	        REGION CATHODE PNP X1 FWD OUTPUT CAM
	            #tempOutputCam ?= #OutputCam.CathodePnPX1FwdOutputCam;
	            #instResetCathodePnPX1FwdOutputCam(Axis := #tempOutputCam^,
	                                               Execute := #statNowCmd = #STAT_RESET,
	                                               Restart:= NOT #tempOutputCam^.StatusWord.%X0);
	        END_REGION

	        REGION CATHODE PNP X1 BWD OUTPUT CAM
	            #tempOutputCam ?= #OutputCam.CathodePnPX1BwdOutputCam;
	            #instResetCathodePnPX1BwdOutputCam(Axis := #tempOutputCam^,
	                                               Execute := #statNowCmd = #STAT_RESET,
	                                               Restart:= NOT #tempOutputCam^.StatusWord.%X0);
	        END_REGION

	        REGION CATHODE PNP X2 FWD OUTPUT CAM
	            #tempOutputCam ?= #OutputCam.CathodePnPX2FwdOutputCam;
	            #instResetCathodePnPX2FwdOutputCam(Axis := #tempOutputCam^,
	                                               Execute := #statNowCmd = #STAT_RESET,
	                                               Restart:= NOT #tempOutputCam^.StatusWord.%X0);
	        END_REGION

	        REGION CATHODE PNP X2 BWD OUTPUT CAM
	            #tempOutputCam ?= #OutputCam.CathodePnPX2BwdOutputCam;
	            #instResetCathodePnPX2BwdOutputCam(Axis := #tempOutputCam^,
	                                               Execute := #statNowCmd = #STAT_RESET,
	                                               Restart:= NOT #tempOutputCam^.StatusWord.%X0);
	        END_REGION

	        REGION CATHODE PNP Z1 DOWN 1 OUTPUT CAM
	            #tempOutputCam ?= #OutputCam.CathodePnPZ1Down1OutputCam;
	            #instResetCathodePnPZ1Down1OutputCam(Axis := #tempOutputCam^,
	                                                 Execute := #statNowCmd = #STAT_RESET,
	                                                 Restart:= NOT #tempOutputCam^.StatusWord.%X0);
	        END_REGION

	        REGION CATHODE PNP Z1 UP 1 OUTPUT CAM
	            #tempOutputCam ?= #OutputCam.CathodePnPZ1Up1OutputCam;
	            #instResetCathodePnPZ1Up1OutputCam(Axis := #tempOutputCam^,
	                                               Execute := #statNowCmd = #STAT_RESET,
	                                               Restart:= NOT #tempOutputCam^.StatusWord.%X0);
	        END_REGION

	        REGION CATHODE PNP Z2 DOWN 1 OUTPUT CAM
	            #tempOutputCam ?= #OutputCam.CathodePnPZ2Down1OutputCam;
	            #instResetCathodePnPZ2Down1OutputCam(Axis := #tempOutputCam^,
	                                                 Execute := #statNowCmd = #STAT_RESET,
	                                                 Restart:= NOT #tempOutputCam^.StatusWord.%X0);
	        END_REGION

	        REGION CATHODE PNP Z2 UP 1 OUTPUT CAM
	            #tempOutputCam ?= #OutputCam.CathodePnPZ2Up1OutputCam;
	            #instResetCathodePnPZ2Up1OutputCam(Axis := #tempOutputCam^,
	                                               Execute := #statNowCmd = #STAT_RESET,
	                                               Restart:= NOT #tempOutputCam^.StatusWord.%X0);
	        END_REGION

	        REGION CATHODE PNP Z1 DOWN 2 OUTPUT CAM
	            #tempOutputCam ?= #OutputCam.CathodePnPZ1Down2OutputCam;
	            #instResetCathodePnPZ1Down2OutputCam(Axis := #tempOutputCam^,
	                                                 Execute := #statNowCmd = #STAT_RESET,
	                                                 Restart:= NOT #tempOutputCam^.StatusWord.%X0);
	        END_REGION

	        REGION CATHODE PNP Z1 UP 2 OUTPUT CAM
	            #tempOutputCam ?= #OutputCam.CathodePnPZ1Up2OutputCam;
	            #instResetCathodePnPZ1Up2OutputCam(Axis := #tempOutputCam^,
	                                               Execute := #statNowCmd = #STAT_RESET,
	                                               Restart:= NOT #tempOutputCam^.StatusWord.%X0);
	        END_REGION

	        REGION CATHODE PNP Z2 DOWN 2 OUTPUT CAM
	            #tempOutputCam ?= #OutputCam.CathodePnPZ2Down2OutputCam;
	            #instResetCathodePnPZ2Down2OutputCam(Axis := #tempOutputCam^,
	                                                 Execute := #statNowCmd = #STAT_RESET,
	                                                 Restart:= NOT #tempOutputCam^.StatusWord.%X0);
	        END_REGION

	        REGION CATHODE PNP Z2 UP 2 OUTPUT CAM
	            #tempOutputCam ?= #OutputCam.CathodePnPZ2Up2OutputCam;
	            #instResetCathodePnPZ2Up2OutputCam(Axis := #tempOutputCam^,
	                                               Execute := #statNowCmd = #STAT_RESET,
	                                               Restart:= NOT #tempOutputCam^.StatusWord.%X0);
	        END_REGION

	        REGION CATHODE PNP Z1 SUCTION ON OUTPUT CAM
	            #tempOutputCam ?= #OutputCam.CathodePnPZ1SuctionOnOutputCam;
	            #instResetCathodePnPZ1SuctionOnOutputCam(Axis := #tempOutputCam^,
	                                                     Execute := #statNowCmd = #STAT_RESET,
	                                                     Restart:= NOT #tempOutputCam^.StatusWord.%X0);
	        END_REGION

	        REGION CATHODE PNP Z1 SUCTION OFF OUTPUT CAM
	            #tempOutputCam ?= #OutputCam.CathodePnPZ1SuctionOffOutputCam;
	            #instResetCathodePnPZ1SuctionOffOutputCam(Axis := #tempOutputCam^,
	                                                      Execute := #statNowCmd = #STAT_RESET,
	                                                      Restart:= NOT #tempOutputCam^.StatusWord.%X0);
	        END_REGION

	        REGION CATHODE PNP Z1 REEL CUT BLOW OUTPUT CAM
	            #tempOutputCam ?= #OutputCam.CathodePnPZ1ReelCutBlowOutputCam;
	            #instResetCathodePnPZ1ReelCutBlowOutputCam(Axis := #tempOutputCam^,
	                                                       Execute := #statNowCmd = #STAT_RESET,
	                                                       Restart:= NOT #tempOutputCam^.StatusWord.%X0);
	        END_REGION

	        REGION CATHODE PNP Z2 SUCTION ON OUTPUT CAM
	            #tempOutputCam ?= #OutputCam.CathodePnPZ2SuctionOnOutputCam;
	            #instResetCathodePnPZ2SuctionOnOutputCam(Axis := #tempOutputCam^,
	                                                     Execute := #statNowCmd = #STAT_RESET,
	                                                     Restart:= NOT #tempOutputCam^.StatusWord.%X0);
	        END_REGION

	        REGION CATHODE PNP Z2 SUCTION OFF OUTPUT CAM
	            #tempOutputCam ?= #OutputCam.CathodePnPZ2SuctionOffOutputCam;
	            #instResetCathodePnPZ2SuctionOffOutputCam(Axis := #tempOutputCam^,
	                                                      Execute := #statNowCmd = #STAT_RESET,
	                                                      Restart:= NOT #tempOutputCam^.StatusWord.%X0);
	        END_REGION

	        REGION CATHODE ALIGN SUCTION ON OUTPUT CAM
	            #tempOutputCam ?= #OutputCam.CathodeAlignSuctionOnOutputCam;
	            #instResetCathodeAlignSuctionOnOutputCam(Axis := #tempOutputCam^,
	                                                     Execute := #statNowCmd = #STAT_RESET,
	                                                     Restart:= NOT #tempOutputCam^.StatusWord.%X0);
	        END_REGION

	        REGION CATHODE ALIGN SUCTION OFF OUTPUT CAM
	            #tempOutputCam ?= #OutputCam.CathodeAlignSuctionOffOutputCam;
	            #instResetCathodeAlignSuctionOffOutputCam(Axis := #tempOutputCam^,
	                                                      Execute := #statNowCmd = #STAT_RESET,
	                                                      Restart:= NOT #tempOutputCam^.StatusWord.%X0);
	        END_REGION

	        REGION FINAL ROLLER X FWD OUTPUT CAM
	            #tempOutputCam ?= #OutputCam.FinalRollerXFwdOutputCam;
	            #instResetFinalRollerXFwdOutputCam(Axis := #tempOutputCam^,
	                                               Execute := #statNowCmd = #STAT_RESET,
	                                               Restart := NOT #tempOutputCam^.StatusWord.%X0);
	        END_REGION

	        REGION FINAL ROLLER X BWD OUTPUT CAM
	            #tempOutputCam ?= #OutputCam.FinalRollerXBwdOutputCam;
	            #instResetFinalRollerXBwdOutputCam(Axis := #tempOutputCam^,
	                                               Execute := #statNowCmd = #STAT_RESET,
	                                               Restart := NOT #tempOutputCam^.StatusWord.%X0);
	        END_REGION

	        REGION FINAL ROLLER X STACK TABLE DOWN OUTPUT CAM
	            #tempOutputCam ?= #OutputCam.FinalRollerXStackTableDownOutputCam;
	            #instResetFinalRollerXStackTableDownOutputCam(Axis := #tempOutputCam^,
	                                                          Execute := #statNowCmd = #STAT_RESET,
	                                                          Restart := NOT #tempOutputCam^.StatusWord.%X0);
	        END_REGION

	        REGION FINAL ROLLER X STACK ANODE VISION OUTPUT CAM
	            #tempOutputCam ?= #OutputCam.FinalRollerXStackAnodeVisionOutputCam;
	            #instResetFinalRollerXStackAnodeVisionOutputCam(Axis := #tempOutputCam^,
	                                                            Execute := #statNowCmd = #STAT_RESET,
	                                                            Restart := NOT #tempOutputCam^.StatusWord.%X0);
	        END_REGION

	        REGION FINAL ROLLER X STACK CATHODE VISION OUTPUT CAM
	            #tempOutputCam ?= #OutputCam.FinalRollerXStackCathodeVisionOutputCam;
	            #instResetFinalRollerXStackCathodeVisionOutputCam(Axis := #tempOutputCam^,
	                                                              Execute := #statNowCmd = #STAT_RESET,
	                                                              Restart := NOT #tempOutputCam^.StatusWord.%X0);
	        END_REGION

	        REGION ANODE PNP Z1 REEL CUT DATA DELETE ON OUTPUT CAM
	            #tempOutputCam ?= #OutputCam.AnodePnPZ1ReelCutDataDeleteOnOutputCam;
	            #instResetAnodePnPZ1ReelCutDataDeleteOnOutputCam(Axis := #tempOutputCam^,
	                                                             Execute := #statNowCmd = #STAT_RESET,
	                                                             Restart := NOT #tempOutputCam^.StatusWord.%X0);
	        END_REGION

	        REGION ANODE PNP 1X REEL CUT DATA DELETE OFF OUTPUT CAM
	            #tempOutputCam ?= #OutputCam.AnodePnP1XReelCutDataDeleteOffOutputCam;
	            #instResetAnodePnP1XReelCutDataDeleteOffOutputCam(Axis := #tempOutputCam^,
	                                                              Execute := #statNowCmd = #STAT_RESET,
	                                                              Restart := NOT #tempOutputCam^.StatusWord.%X0);
	        END_REGION

	        REGION ANODE ALIGN VISION OUTPUT CAM
	            #tempOutputCam ?= #OutputCam.AnodeAlignVisionOutputCam;
	            #instResetAnodeAlignVisionOutputCam(Axis := #tempOutputCam^,
	                                                Execute := #statNowCmd = #STAT_RESET,
	                                                Restart := NOT #tempOutputCam^.StatusWord.%X0);
	        END_REGION

	        REGION CATHODE PNP Z1 REEL CUT DATA DELETE ON OUTPUT CAM
	            #tempOutputCam ?= #OutputCam.CathodePnPZ1ReelCutDataDeleteOnOutputCam;
	            #instResetCathodePnPZ1ReelCutDataDeleteOnOutputCam(Axis := #tempOutputCam^,
	                                                               Execute := #statNowCmd = #STAT_RESET,
	                                                               Restart := NOT #tempOutputCam^.StatusWord.%X0);
	        END_REGION

	        REGION CATHODE PNP 1X REEL CUT DATA DELETE OFF OUTPUT CAM
	            #tempOutputCam ?= #OutputCam.CathodePnP1XReelCutDataDeleteOffOutputCam;
	            #instResetCathodePnP1XReelCutDataDeleteOffOutputCam(Axis := #tempOutputCam^,
	                                                                Execute := #statNowCmd = #STAT_RESET,
	                                                                Restart := NOT #tempOutputCam^.StatusWord.%X0);
	        END_REGION

	        REGION CATHODE ALIGN VISION OUTPUT CAM
	            #tempOutputCam ?= #OutputCam.CathodeAlignVisionOutputCam;
	            #instResetCathodeAlignVisionOutputCam(Axis := #tempOutputCam^,
	                                                  Execute := #statNowCmd = #STAT_RESET,
	                                                  Restart := NOT #tempOutputCam^.StatusWord.%X0);
	        END_REGION

	    END_REGION
	END_REGION

	REGION OUTPUT SIGNAL                                                                    // 각 커맨드 동작 시 상태 표시 출력
	    #Busy := #statNowCmd = #STAT_START
	    OR #statNowCmd = #STAT_RESET;
	    #Done := #statNowCmd = #STAT_DONE;
	    #Error := #statNowCmd = #STAT_ERROR;
	    #NowCmd := #statNowCmd;
	    #BeforeCmd := #statBeforeCmd;
	END_REGION

END_FUNCTION_BLOCK

